{attribute 'enable_dynamic_creation'}
FUNCTION_BLOCK INTERNAL FB_XmlLogger IMPLEMENTS ILogger
VAR_INPUT
END_VAR
VAR_OUTPUT
END_VAR
VAR
END_VAR

METHOD PUBLIC Write : STRING
VAR_INPUT
	sMsg	: string;
END_VAR
Write := CONCAT('XmlLogger: ', sMsg);
END_METHOD

END_FUNCTION_BLOCK

(* stored: Version 1.1.0.1, ProductVersion 3.1.4024.12
   POU FB_XmlLogger: Id {723c9ffc-e38d-49bc-b062-716cfc1f7baf}, SpecialFunc None
   Method Write: Id {2db2e170-93d8-4538-b6b2-a82a0d9d5c99} *)
